TYPE EcCoeSdoWrite_Status_typ :
	STRUCT
		bBusy           : BOOL;
        bError          : BOOL;
	END_STRUCT
END_TYPE

(* stored: Version 1.1.0.1, ProductVersion 3.1.4024.3
   DUT EcCoeSdoWrite_Status_typ: Id {455719d7-7639-0fa9-322c-382f3566cf13} *)
